(* PLC project TwinForgeImportTest2.project, CODESYS CODESYS V3.5 SP22 Patch 2 *)
(* stored: creationDateTime 2026-07-23T18:26:45.620772, modificationDateTime 2026-07-23T18:11:10.4936387 *)

PROGRAM PLC_PRG
  VAR
    xStartBtn : BOOL;
    xMotorOnOff : BOOL;
  END_VAR

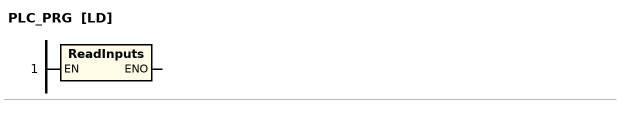
(* LD diagram, written out as Structured Text *)

ReadInputs();

ACTION ReadInputs:
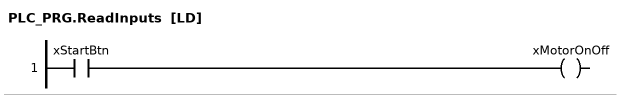
(* LD diagram, written out as Structured Text *)

xMotorOnOff := xStartBtn;
END_ACTION
END_PROGRAM

CONFIGURATION Application
  RESOURCE Application ON PLC
    TASK MainTask(INTERVAL := T#20ms, PRIORITY := 1);
    PROGRAM PLC_PRG WITH MainTask : PLC_PRG;
  END_RESOURCE
END_CONFIGURATION
